FUNCTION_BLOCK EmergencyDecideInit (* Basic Function Block Type *)
  (* Standard: 61499-2 *)
  (* Version 0.0, 7/15/2026, Schneider Electric, Template *)
  PACKAGE SE.Nereda;
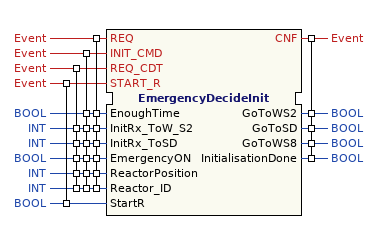
  EVENT_INPUT
    REQ WITH EnoughTime, InitRx_ToW_S2, InitRx_ToSD, Reactor_ID, EmergencyON, ReactorPosition; (* Normal Execution Request *)
    INIT_CMD WITH EmergencyON, EnoughTime, InitRx_ToW_S2, InitRx_ToSD, Reactor_ID, ReactorPosition;
    REQ_CDT WITH InitRx_ToW_S2, InitRx_ToSD, Reactor_ID, EmergencyON, ReactorPosition;
    START_R WITH StartR;
  END_EVENT
  EVENT_OUTPUT
    CNF WITH GoToSD, GoToWS8, InitialisationDone, GoToWS2; (* Execution Confirmation *)
  END_EVENT
  VAR_INPUT
    EnoughTime : BOOL; (* Input event qualifier *)
    InitRx_ToW_S2 : INT;
    InitRx_ToSD : INT;
    EmergencyON : BOOL;
    ReactorPosition : INT;
    Reactor_ID : INT;
    StartR : BOOL;
  END_VAR
  VAR_OUTPUT
    GoToWS2 : BOOL;
    GoToSD : BOOL; (* Output event qualifier *)
    GoToWS8 : BOOL;
    InitialisationDone : BOOL;
  END_VAR
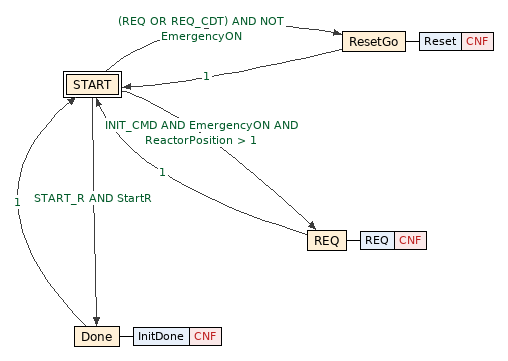
  EC_STATES
    START; (* Initial State *)
    REQ : REQ -> CNF; (* Normal execution *)
    ResetGo : Reset -> CNF;
    Done : InitDone -> CNF;
  END_STATES
  EC_TRANSITIONS
    START TO REQ := INIT_CMD AND EmergencyON AND ReactorPosition > 1;
    REQ TO START := 1;
    START TO ResetGo := (REQ OR REQ_CDT) AND NOT EmergencyON;
    ResetGo TO START := 1;
    START TO Done := START_R AND StartR;
    Done TO START := 1;
  END_TRANSITIONS
  ALGORITHM REQ IN ST: (* Normally executed algorithm *)
;
IF EnoughTime THEN
	GoToWS8 := FALSE;
	InitialisationDone := FALSE;
	IF InitRx_ToW_S2 = Reactor_ID THEN
		GoToSD := FALSE;
		GoToWS2 := TRUE;
	ELSIF InitRx_ToSD = Reactor_ID THEN
		GoToSD := TRUE;
		GoToWS2 := FALSE;
	END_IF;
ELSE
	GoToSD := FALSE;
	GoToWS2 := FALSE;
	GoToWS8 := TRUE;
	InitialisationDone := FALSE;
END_IF;
  END_ALGORITHM
  ALGORITHM Reset IN ST:
;
GoToSD := FALSE;
GoToWS2 := FALSE;
GoToWS8 := FALSE;
  END_ALGORITHM
  ALGORITHM InitDone IN ST:
;
GoToSD := FALSE;
GoToWS2 := FALSE;
GoToWS8 := FALSE;
InitialisationDone := TRUE;
  END_ALGORITHM
END_FUNCTION_BLOCK
